PROGRAM MAIN
VAR
END_VAR

END_PROGRAM

(* stored: Version 1.1.0.1
   POU MAIN: Id {b5d42716-8ce5-440e-8a1d-b0c25a730ea8} *)
